// TIA Portal V17 export
// export: Created 2023-02-13T11:16:52.4672257Z, ExportSetting WithDefaults, DisplayName Totally Integrated Automation Portal, DisplayVersion V17, DisplayName TIA Portal Openness, DisplayVersion V17, DisplayName TIA Portal Teamcenter Gateway, DisplayVersion V17, DisplayName TIA Portal Version Control Interface, DisplayVersion V17, DisplayName SINAMICS Startdrive Advanced, DisplayVersion V17, DisplayName SINAMICS Startdrive G130, G150, S120, S150, SINAMICS MV, S210, DisplayVersion V17, DisplayName SINAMICS Startdrive G110M, G120, G120C, G120D, G120P, G115D, DisplayVersion V17, DisplayName STEP 7 Professional, DisplayVersion V17, DisplayName STEP 7 Safety, DisplayVersion V17, DisplayName WinCC Professional, DisplayVersion V17
DATA_BLOCK "Gen_Line_Prep"   // DB36
{ S7_Optimized_Access := 'TRUE' }
VERSION : 0.1
// stored: AutoNumber true, DBAccessibleFromOPCUA true, DBAccessibleFromWebserver true, IsOnlyStoredInLoadMemory false, IsRetainMemResEnabled false, IsWriteProtectedInAS false, MemoryReserve 100
   VAR
      T09_Line : Struct
         "AV-09_01" : Bool;
         "AV-09_2" : Bool;
         "AV-09_3" : Bool;
         "AV-09_4" : Bool;
         "AV-09_5" : Bool;
         "AV-09_6" : Bool;
         "AV-09_7" : Bool;
         "AV-09_8" : Bool;
         "AV-09_9" : Bool;
         "AV-09_10" : Bool;
         "P-09.01" : Bool;
         "P-09.2" : Bool;
         "P-09.3" : Bool;
         Line_Prod : Bool;
      END_STRUCT;
      Gen_Garlic_Vinegar : Struct
         Line_Pro_Water : Bool;
      END_STRUCT;
   END_VAR
BEGIN
END_DATA_BLOCK
